INTERFACE INTERNAL ITF_1_Skill EXTENDS ITF_0_BaseComponent

PROPERTY Busy : BOOL
GET
END_GET
END_PROPERTY

PROPERTY Done : BOOL
GET
END_GET
END_PROPERTY

METHOD INTERNAL Pause : BOOL
VAR_INPUT
END_VAR
END_METHOD

METHOD INTERNAL Restart : BOOL
VAR_INPUT
END_VAR
END_METHOD

METHOD INTERNAL Resume : BOOL
VAR_INPUT
END_VAR
END_METHOD

METHOD INTERNAL Start : BOOL
VAR_INPUT
END_VAR
END_METHOD

METHOD INTERNAL Stop : BOOL
VAR_INPUT
END_VAR
END_METHOD

END_INTERFACE

(* stored: Version 1.1.0.1, ProductVersion 3.1.4026.18
   Itf ITF_1_Skill: Id {f4c05153-2d3e-4022-88ce-5221103f1d43}
   Property Busy: Id {51aed81e-bfa5-49ca-a544-38e4c63eea80}
   Get Get: Id {9c2f2cc4-b1d5-4ed2-922c-6495bbd4ed95}
   Property Done: Id {9eaff107-3cf8-498a-ae76-6575db90152c}
   Get Get: Id {1c046abe-d464-4663-8f78-42669896567b}
   Method Pause: Id {c803a7d8-124f-43ed-8711-bf61a5121e40}
   Method Restart: Id {d8486a93-cc8f-4854-a88f-32d43fe5817e}
   Method Resume: Id {3004afec-1d0b-4787-b759-23c588507fa4}
   Method Start: Id {a5bff2ad-fde8-4853-845d-6c29ed141111}
   Method Stop: Id {747ee5b7-7cb0-4f9d-a367-37335edac648} *)
